(* IEC 61131-3 sources: plc_on_fpga_riscv_hybrid/RV_FPGA_PLC_IDE_Projects/Comparison_Test, 1 file *)

(* ---- Comparison_Test.il ---- *)
VAR
END_VAR

PROGRAM Comparison_Test
    Less_Than :
        LD     25
        LT     5
        ST     %LEDG.0
END_PROGRAM
